# EPICS autosave request: GeRM-192/Mars_DDM/iocBoot/ioczDDM/auto_settings.req
file "hera_settings.req"
file "hera_array+settings.req"
